TYPE LG_Statusbits :
STRUCT
	b_WaterFlowNOK				:	BOOL;
	b_WaterPumpOn				:	BOOL;
	b_ExtWaterPumpOn			:	BOOL;
	b_CompressorOn				:	BOOL;
	b_DefrostOn					:	BOOL;
	b_SWWModeOn					:	BOOL;
	b_SWWTankDesinfectionActive	:	BOOL;
	b_SilentModeOn				:	BOOL;
	b_CoolingActive				:	BOOL;
	b_SolarPumpActive			:	BOOL;
	b_BackupHeater1Active		:	BOOL;
	b_BackupHeater2Active		:	BOOL;
	b_SWWBoostHeaterActive		:	BOOL;
	b_ErrorActive				:	BOOL;
	b_EMOperationAvailable		:	BOOL;
	b_EMSWWOperationAvailable	:	BOOL;
	b_MixPumpActive				:	BOOL;
	
END_STRUCT
END_TYPE

(* stored: Version 1.1.0.1, ProductVersion 3.1.4026.18
   DUT LG_Statusbits: Id {71abbfda-afa9-4e86-9891-5f164d391cb3} *)
